// TIA Portal V17 export
// export: Created 2025-05-22T06:01:04.2194425Z, ExportSetting WithDefaults, DisplayName Totally Integrated Automation Portal, DisplayVersion V17 Update 8, DisplayName TIA Portal Openness, DisplayVersion V17 Update 8, DisplayName TIA Portal Version Control Interface, DisplayVersion V17, DisplayName SINAMICS Startdrive Advanced, DisplayVersion V17 SP2, DisplayName SINAMICS Startdrive G110M, G120, G120C, G120D, G120P, G115D, DisplayVersion V17 SP2, DisplayName SINAMICS Startdrive G130, G150, S120, S150, SINAMICS MV, S210, DisplayVersion V17 SP2, DisplayName STEP 7 Professional, DisplayVersion V17 Update 8, DisplayName SINUMERIK ONE STEP 7 Toolbox, DisplayVersion V17 Update 12, DisplayName SINUMERIK ONE PLC Basic Program Plus, DisplayVersion V17 Update 12, DisplayName SINUMERIK 840D sl STEP 7 Toolbox, DisplayVersion V17 Update 12, DisplayName STEP 7 Safety, DisplayVersion V17 Update 6, DisplayName WinCC Advanced, DisplayVersion V17 Update 8
DATA_BLOCK "DB2100_GENERAL"   // DB2100
{ S7_Optimized_Access := 'FALSE'; DB_Accessible_From_OPC_UA := 'FALSE' }
AUTHOR : ETXETAR
VERSION : 1.0
// stored: AutoNumber false, DBAccessibleFromOPCUA false, DBAccessibleFromWebserver true, IsOnlyStoredInLoadMemory false, IsWriteProtectedInAS false
   VAR RETAIN
      EMERGENCY_STOP_ACTIVE : Bool;   // EMERGENCY STOP PILZ / EMERGENCY STOP ACTIVE
      SAFETY_GATES_CLOSED_LOCKED : Bool;   // GATES CLOSED & LOCKED PILZ / SAFETY GATES CLOSED AND LOCKED
      MACHINE_READY_POWER_ENABLED : Bool;   // MACHINE READY PILZ / MACHINE READY POWER ENABLED
      ANY_AXIS_OR_CH_BYPASSED : Bool;   // ANY AXIS BYPASSED / ANY AXIS OR CHANNEL BYPASSED
      ANY_AXIS_OR_CH_BYPASSED_ALARM : Bool;   // ANY AXIS BYPASSED FAULT / ANY AXIS OR CHANNEL BYPASSED ALARM
      PROGRAMMING_ALARM : Bool;   // ANY PROGRAMMING ALARM
      CHECKSUM_OK : Bool;   // CITI Checksum Overall OK / CHECKSUM OK
      EMERGENCY_STOP_ACTIVE_ALARM : Bool;   // EMERGENCY STOP ACTIVE / EMERGENCY STOP ACTIVE ALARM
      OVERRIDE_LOWER_THAN_80 : Bool;   // OVERRIDE LOWER THAN 80
      OVERRIDE_100 : Bool;   // OVERRIDE 100
      WARNINGS_GONE : Bool;   // UTILITY SKIDS WARNINGS GONE
      CHECK_NETWORK_LOGIC_ALARM : Bool;   // CHECK NETWORK LOGIC ALARM
      U01_SAFETY_GATES_CLOSED_LOCKED : Bool;   // UNIT 01 SAFETY GATES CLOSED AND LOCKED
      U02_SAFETY_GATES_CLOSED_LOCKED : Bool;   // UNIT 02 SAFETY GATES CLOSED AND LOCKED
      AXIS_Z13_ENABLED_DELAYED_AUX : Bool;   // AXIS Z13 ENABLED DELAYED AUXILIARY
      AXIS_Z23_ENABLED_DELAYED_AUX : Bool;   // AXIS Z23 ENABLED DELAYED AUXILIARY
   END_VAR
BEGIN
END_DATA_BLOCK
